Universal Robots URScript: A_penguin.script

def draw_penguin():
  # --- Robot Setup (ADJUST THESE VALUES) ---
  # Base position for the drawing (e.g., center of the A4 paper in robot's reach)
  base_p = p[0.4, -0.2, 0.2, 2.22, -2.22, 0]

  # Set the TCP for your marker tip. E.g., p[0, 0, 0.15, 0, 0, 0] for a 15cm offset
  # set_tcp(p[0, 0, 0.15, 0, 0, 0])

  # Movement parameters
  vel = 0.075
  accel = 0.1

  # Z heights for drawing (on paper) and moving (lifted)
  z_draw = base_p[2] - 0.005 # Adjust this based on paper height
  z_move = base_p[2] + 0.020 # 2cm lift

  # --- Drawing Logic ---
  textmsg("Starting the drawing process")
\n  # --- Path 1 ---\n  movel(pose(base_p[0] + 0.16907999999999998, base_p[1] + 0.024779999999999986, z_move, base_p[3], base_p[4], base_p[5]), a=accel, v=vel)\n  movel(pose(base_p[0] + 0.16907999999999998, base_p[1] + 0.024779999999999986, z_draw, base_p[3], base_p[4], base_p[5]), a=accel, v=vel)\n  movel(pose(base_p[0] + 0.1716, base_p[1] + 0.024779999999999986, z_draw, base_p[3], base_p[4], base_p[5]), a=accel, v=vel)\n  movel(pose(base_p[0] + 0.1716, base_p[1] + 0.024779999999999986, z_move, base_p[3], base_p[4], base_p[5]), a=accel, v=vel)\n\n  # --- Path 2 ---\n  movel(pose(base_p[0] + 0.18419999999999997, base_p[1] + 0.025619999999999987, z_move, base_p[3], base_p[4], base_p[5]), a=accel, v=vel)\n  movel(pose(base_p[0] + 0.18419999999999997, base_p[1] + 0.025619999999999987, z_draw, base_p[3], base_p[4], base_p[5]), a=accel, v=vel)\n  movel(pose(base_p[0] + 0.18336000000000002, base_p[1] + 0.024779999999999986, z_draw, base_p[3], base_p[4], base_p[5]), a=accel, v=vel)\n  movel(pose(base_p[0] + 0.18084, base_p[1] + 0.024779999999999986, z_draw, base_p[3], base_p[4], base_p[5]), a=accel, v=vel)\n  movel(pose(base_p[0] + 0.18419999999999997, base_p[1] + 0.024779999999999986, z_draw, base_p[3], base_p[4], base_p[5]), a=accel, v=vel)\n  movel(pose(base_p[0] + 0.18419999999999997, base_p[1] + 0.024779999999999986, z_move, base_p[3], base_p[4], base_p[5]), a=accel, v=vel)\n\n  # --- Path 3 ---\n  movel(pose(base_p[0] + 0.11279999999999998, base_p[1] + 0.025619999999999987, z_move, base_p[3], base_p[4], base_p[5]), a=accel, v=vel)\n  movel(pose(base_p[0] + 0.11279999999999998, base_p[1] + 0.025619999999999987, z_draw, base_p[3], base_p[4], base_p[5]), a=accel, v=vel)\n  movel(pose(base_p[0] + 0.11279999999999998, base_p[1] + 0.024779999999999986, z_draw, base_p[3], base_p[4], base_p[5]), a=accel, v=vel)\n  movel(pose(base_p[0] + 0.11363999999999999, base_p[1] + 0.023939999999999986, z_draw, base_p[3], base_p[4], base_p[5]), a=accel, v=vel)\n  movel(pose(base_p[0] + 0.11447999999999998, base_p[1] + 0.024779999999999986, z_draw, base_p[3], base_p[4], base_p[5]), a=accel, v=vel)\n  movel(pose(base_p[0] + 0.11616, base_p[1] + 0.024779999999999986, z_draw, base_p[3], base_p[4], base_p[5]), a=accel, v=vel)\n  movel(pose(base_p[0] + 0.11363999999999999, base_p[1] + 0.024779999999999986, z_draw, base_p[3], base_p[4], base_p[5]), a=accel, v=vel)\n  movel(pose(base_p[0] + 0.11363999999999999, base_p[1] + 0.024779999999999986, z_move, base_p[3], base_p[4], base_p[5]), a=accel, v=vel)\n\n  # --- Path 4 ---\n  movel(pose(base_p[0] + 0.16572, base_p[1] + 0.03401999999999999, z_move, base_p[3], base_p[4], base_p[5]), a=accel, v=vel)\n  movel(pose(base_p[0] + 0.16572, base_p[1] + 0.03401999999999999, z_draw, base_p[3], base_p[4], base_p[5]), a=accel, v=vel)\n  movel(pose(base_p[0] + 0.16656, base_p[1] + 0.033179999999999994, z_draw, base_p[3], base_p[4], base_p[5]), a=accel, v=vel)\n  movel(pose(base_p[0] + 0.17244, base_p[1] + 0.033179999999999994, z_draw, base_p[3], base_p[4], base_p[5]), a=accel, v=vel)\n  movel(pose(base_p[0] + 0.17244, base_p[1] + 0.03401999999999999, z_draw, base_p[3], base_p[4], base_p[5]), a=accel, v=vel)\n  movel(pose(base_p[0] + 0.1716, base_p[1] + 0.033179999999999994, z_draw, base_p[3], base_p[4], base_p[5]), a=accel, v=vel)\n  movel(pose(base_p[0] + 0.16739999999999997, base_p[1] + 0.033179999999999994, z_draw, base_p[3], base_p[4], base_p[5]), a=accel, v=vel)\n  movel(pose(base_p[0] + 0.16656, base_p[1] + 0.03401999999999999, z_draw, base_p[3], base_p[4], base_p[5]), a=accel, v=vel)\n  movel(pose(base_p[0] + 0.16824, base_p[1] + 0.03569999999999999, z_draw, base_p[3], base_p[4], base_p[5]), a=accel, v=vel)\n  movel(pose(base_p[0] + 0.16992000000000002, base_p[1] + 0.03569999999999999, z_draw, base_p[3], base_p[4], base_p[5]), a=accel, v=vel)\n  movel(pose(base_p[0] + 0.17076, base_p[1] + 0.03485999999999999, z_draw, base_p[3], base_p[4], base_p[5]), a=accel, v=vel)\n  movel(pose(base_p[0] + 0.1716, base_p[1] + 0.03569999999999999, z_draw, base_p[3], base_p[4], base_p[5]), a=accel, v=vel)\n  movel(pose(base_p[0] + 0.17412, base_p[1] + 0.03569999999999999, z_draw, base_p[3], base_p[4], base_p[5]), a=accel, v=vel)\n  movel(pose(base_p[0] + 0.16824, base_p[1] + 0.03569999999999999, z_draw, base_p[3], base_p[4], base_p[5]), a=accel, v=vel)\n  movel(pose(base_p[0] + 0.16739999999999997, base_p[1] + 0.03485999999999999, z_draw, base_p[3], base_p[4], base_p[5]), a=accel, v=vel)\n  movel(pose(base_p[0] + 0.16656, base_p[1] + 0.03485999999999999, z_draw, base_p[3], base_p[4], base_p[5]), a=accel, v=vel)\n  movel(pose(base_p[0] + 0.16656, base_p[1] + 0.03485999999999999, z_move, base_p[3], base_p[4], base_p[5]), a=accel, v=vel)\n\n  # --- Path 5 ---\n  movel(pose(base_p[0] + 0.12372, base_p[1] + 0.03653999999999999, z_move, base_p[3], base_p[4], base_p[5]), a=accel, v=vel)\n  movel(pose(base_p[0] + 0.12372, base_p[1] + 0.03653999999999999, z_draw, base_p[3], base_p[4], base_p[5]), a=accel, v=vel)\n  movel(pose(base_p[0] + 0.12455999999999999, base_p[1] + 0.03569999999999999, z_draw, base_p[3], base_p[4], base_p[5]), a=accel, v=vel)\n  movel(pose(base_p[0] + 0.12624, base_p[1] + 0.03569999999999999, z_draw, base_p[3], base_p[4], base_p[5]), a=accel, v=vel)\n  movel(pose(base_p[0] + 0.12708, base_p[1] + 0.03485999999999999, z_draw, base_p[3], base_p[4], base_p[5]), a=accel, v=vel)\n  movel(pose(base_p[0] + 0.1296, base_p[1] + 0.03485999999999999, z_draw, base_p[3], base_p[4], base_p[5]), a=accel, v=vel)\n  movel(pose(base_p[0] + 0.13127999999999998, base_p[1] + 0.033179999999999994, z_draw, base_p[3], base_p[4], base_p[5]), a=accel, v=vel)\n  movel(pose(base_p[0] + 0.13044, base_p[1] + 0.03233999999999999, z_draw, base_p[3], base_p[4], base_p[5]), a=accel, v=vel)\n  movel(pose(base_p[0] + 0.12791999999999998, base_p[1] + 0.03233999999999999, z_draw, base_p[3], base_p[4], base_p[5]), a=accel, v=vel)\n  movel(pose(base_p[0] + 0.12708, base_p[1] + 0.033179999999999994, z_draw, base_p[3], base_p[4], base_p[5]), a=accel, v=vel)\n  movel(pose(base_p[0] + 0.12624, base_p[1] + 0.03233999999999999, z_draw, base_p[3], base_p[4], base_p[5]), a=accel, v=vel)\n  movel(pose(base_p[0] + 0.12539999999999998, base_p[1] + 0.033179999999999994, z_draw, base_p[3], base_p[4], base_p[5]), a=accel, v=vel)\n  movel(pose(base_p[0] + 0.12455999999999999, base_p[1] + 0.033179999999999994, z_draw, base_p[3], base_p[4], base_p[5]), a=accel, v=vel)\n  movel(pose(base_p[0] + 0.12539999999999998, base_p[1] + 0.033179999999999994, z_draw, base_p[3], base_p[4], base_p[5]), a=accel, v=vel)\n  movel(pose(base_p[0] + 0.12624, base_p[1] + 0.03233999999999999, z_draw, base_p[3], base_p[4], base_p[5]), a=accel, v=vel)\n  movel(pose(base_p[0] + 0.12708, base_p[1] + 0.033179999999999994, z_draw, base_p[3], base_p[4], base_p[5]), a=accel, v=vel)\n  movel(pose(base_p[0] + 0.12791999999999998, base_p[1] + 0.03233999999999999, z_draw, base_p[3], base_p[4], base_p[5]), a=accel, v=vel)\n  movel(pose(base_p[0] + 0.13127999999999998, base_p[1] + 0.03233999999999999, z_draw, base_p[3], base_p[4], base_p[5]), a=accel, v=vel)\n  movel(pose(base_p[0] + 0.13127999999999998, base_p[1] + 0.03401999999999999, z_draw, base_p[3], base_p[4], base_p[5]), a=accel, v=vel)\n  movel(pose(base_p[0] + 0.13044, base_p[1] + 0.03401999999999999, z_draw, base_p[3], base_p[4], base_p[5]), a=accel, v=vel)\n  movel(pose(base_p[0] + 0.1296, base_p[1] + 0.03485999999999999, z_draw, base_p[3], base_p[4], base_p[5]), a=accel, v=vel)\n  movel(pose(base_p[0] + 0.12708, base_p[1] + 0.03485999999999999, z_draw, base_p[3], base_p[4], base_p[5]), a=accel, v=vel)\n  movel(pose(base_p[0] + 0.12624, base_p[1] + 0.03569999999999999, z_draw, base_p[3], base_p[4], base_p[5]), a=accel, v=vel)\n  movel(pose(base_p[0] + 0.12539999999999998, base_p[1] + 0.03569999999999999, z_draw, base_p[3], base_p[4], base_p[5]), a=accel, v=vel)\n  movel(pose(base_p[0] + 0.12455999999999999, base_p[1] + 0.03653999999999999, z_draw, base_p[3], base_p[4], base_p[5]), a=accel, v=vel)\n  movel(pose(base_p[0] + 0.12455999999999999, base_p[1] + 0.03653999999999999, z_move, base_p[3], base_p[4], base_p[5]), a=accel, v=vel)\n\n  # --- Path 6 ---\n  movel(pose(base_p[0] + 0.13883999999999996, base_p[1] + 0.040739999999999985, z_move, base_p[3], base_p[4], base_p[5]), a=accel, v=vel)\n  movel(pose(base_p[0] + 0.13883999999999996, base_p[1] + 0.040739999999999985, z_draw, base_p[3], base_p[4], base_p[5]), a=accel, v=vel)\n  movel(pose(base_p[0] + 0.13968, base_p[1] + 0.03989999999999999, z_draw, base_p[3], base_p[4], base_p[5]), a=accel, v=vel)\n  movel(pose(base_p[0] + 0.13968, base_p[1] + 0.03905999999999999, z_draw, base_p[3], base_p[4], base_p[5]), a=accel, v=vel)\n  movel(pose(base_p[0] + 0.14051999999999998, base_p[1] + 0.03905999999999999, z_draw, base_p[3], base_p[4], base_p[5]), a=accel, v=vel)\n  movel(pose(base_p[0] + 0.14136, base_p[1] + 0.03821999999999998, z_draw, base_p[3], base_p[4], base_p[5]), a=accel, v=vel)\n  movel(pose(base_p[0] + 0.14304, base_p[1] + 0.03821999999999998, z_draw, base_p[3], base_p[4], base_p[5]), a=accel, v=vel)\n  movel(pose(base_p[0] + 0.14388, base_p[1] + 0.03737999999999999, z_draw, base_p[3], base_p[4], base_p[5]), a=accel, v=vel)\n  movel(pose(base_p[0] + 0.14472, base_p[1] + 0.03737999999999999, z_draw, base_p[3], base_p[4], base_p[5]), a=accel, v=vel)\n  movel(pose(base_p[0] + 0.14556, base_p[1] + 0.03653999999999999, z_draw, base_p[3], base_p[4], base_p[5]), a=accel, v=vel)\n  movel(pose(base_p[0] + 0.14639999999999997, base_p[1] + 0.03737999999999999, z_draw, base_p[3], base_p[4], base_p[5]), a=accel, v=vel)\n  movel(pose(base_p[0] + 0.14724, base_p[1] + 0.03737999999999999, z_draw, base_p[3], base_p[4], base_p[5]), a=accel, v=vel)\n  movel(pose(base_p[0] + 0.14808, base_p[1] + 0.03653999999999999, z_draw, base_p[3], base_p[4], base_p[5]), a=accel, v=vel)\n  movel(pose(base_p[0] + 0.14976, base_p[1] + 0.03653999999999999, z_draw, base_p[3], base_p[4], base_p[5]), a=accel, v=vel)\n  movel(pose(base_p[0] + 0.15059999999999998, base_p[1] + 0.03737999999999999, z_draw, base_p[3], base_p[4], base_p[5]), a=accel, v=vel)\n  movel(pose(base_p[0] + 0.15228, base_p[1] + 0.03737999999999999, z_draw, base_p[3], base_p[4], base_p[5]), a=accel, v=vel)\n  movel(pose(base_p[0] + 0.15312, base_p[1] + 0.03821999999999998, z_draw, base_p[3], base_p[4], base_p[5]), a=accel, v=vel)\n  movel(pose(base_p[0] + 0.15395999999999999, base_p[1] + 0.03821999999999998, z_draw, base_p[3], base_p[4], base_p[5]), a=accel, v=vel)\n  movel(pose(base_p[0] + 0.15480000000000002, base_p[1] + 0.03905999999999999, z_draw, base_p[3], base_p[4], base_p[5]), a=accel, v=vel)\n  movel(pose(base_p[0] + 0.15563999999999997, base_p[1] + 0.03905999999999999, z_draw, base_p[3], base_p[4], base_p[5]), a=accel, v=vel)\n  movel(pose(base_p[0] + 0.15647999999999998, base_p[1] + 0.03989999999999999, z_draw, base_p[3], base_p[4], base_p[5]), a=accel, v=vel)\n  movel(pose(base_p[0] + 0.15563999999999997, base_p[1] + 0.03989999999999999, z_draw, base_p[3], base_p[4], base_p[5]), a=accel, v=vel)\n  movel(pose(base_p[0] + 0.15480000000000002, base_p[1] + 0.03905999999999999, z_draw, base_p[3], base_p[4], base_p[5]), a=accel, v=vel)\n  movel(pose(base_p[0] + 0.15395999999999999, base_p[1] + 0.03905999999999999, z_draw, base_p[3], base_p[4], base_p[5]), a=accel, v=vel)\n  movel(pose(base_p[0] + 0.15228, base_p[1] + 0.03737999999999999, z_draw, base_p[3], base_p[4], base_p[5]), a=accel, v=vel)\n  movel(pose(base_p[0] + 0.15059999999999998, base_p[1] + 0.03737999999999999, z_draw, base_p[3], base_p[4], base_p[5]), a=accel, v=vel)\n  movel(pose(base_p[0] + 0.14976, base_p[1] + 0.03653999999999999, z_draw, base_p[3], base_p[4], base_p[5]), a=accel, v=vel)\n  movel(pose(base_p[0] + 0.14808, base_p[1] + 0.03653999999999999, z_draw, base_p[3], base_p[4], base_p[5]), a=accel, v=vel)\n  movel(pose(base_p[0] + 0.14724, base_p[1] + 0.03737999999999999, z_draw, base_p[3], base_p[4], base_p[5]), a=accel, v=vel)\n  movel(pose(base_p[0] + 0.14472, base_p[1] + 0.03737999999999999, z_draw, base_p[3], base_p[4], base_p[5]), a=accel, v=vel)\n  movel(pose(base_p[0] + 0.14388, base_p[1] + 0.03821999999999998, z_draw, base_p[3], base_p[4], base_p[5]), a=accel, v=vel)\n  movel(pose(base_p[0] + 0.14136, base_p[1] + 0.03821999999999998, z_draw, base_p[3], base_p[4], base_p[5]), a=accel, v=vel)\n  movel(pose(base_p[0] + 0.13968, base_p[1] + 0.03989999999999999, z_draw, base_p[3], base_p[4], base_p[5]), a=accel, v=vel)\n  movel(pose(base_p[0] + 0.13968, base_p[1] + 0.040739999999999985, z_draw, base_p[3], base_p[4], base_p[5]), a=accel, v=vel)\n  movel(pose(base_p[0] + 0.13968, base_p[1] + 0.040739999999999985, z_move, base_p[3], base_p[4], base_p[5]), a=accel, v=vel)\n\n  # --- Path 7 ---\n  movel(pose(base_p[0] + 0.09348, base_p[1] + 0.11045999999999999, z_move, base_p[3], base_p[4], base_p[5]), a=accel, v=vel)\n  movel(pose(base_p[0] + 0.09348, base_p[1] + 0.11045999999999999, z_draw, base_p[3], base_p[4], base_p[5]), a=accel, v=vel)\n  movel(pose(base_p[0] + 0.09011999999999999, base_p[1] + 0.10878, z_draw, base_p[3], base_p[4], base_p[5]), a=accel, v=vel)\n  movel(pose(base_p[0] + 0.08675999999999999, base_p[1] + 0.10542, z_draw, base_p[3], base_p[4], base_p[5]), a=accel, v=vel)\n  movel(pose(base_p[0] + 0.08591999999999998, base_p[1] + 0.10289999999999999, z_draw, base_p[3], base_p[4], base_p[5]), a=accel, v=vel)\n  movel(pose(base_p[0] + 0.07919999999999999, base_p[1] + 0.09617999999999999, z_draw, base_p[3], base_p[4], base_p[5]), a=accel, v=vel)\n  movel(pose(base_p[0] + 0.07835999999999999, base_p[1] + 0.09617999999999999, z_draw, base_p[3], base_p[4], base_p[5]), a=accel, v=vel)\n  movel(pose(base_p[0] + 0.07499999999999998, base_p[1] + 0.09029999999999999, z_draw, base_p[3], base_p[4], base_p[5]), a=accel, v=vel)\n  movel(pose(base_p[0] + 0.07247999999999999, base_p[1] + 0.08777999999999998, z_draw, base_p[3], base_p[4], base_p[5]), a=accel, v=vel)\n  movel(pose(base_p[0] + 0.06828, base_p[1] + 0.07937999999999999, z_draw, base_p[3], base_p[4], base_p[5]), a=accel, v=vel)\n  movel(pose(base_p[0] + 0.06828, base_p[1] + 0.07769999999999999, z_draw, base_p[3], base_p[4], base_p[5]), a=accel, v=vel)\n  movel(pose(base_p[0] + 0.07247999999999999, base_p[1] + 0.08694, z_draw, base_p[3], base_p[4], base_p[5]), a=accel, v=vel)\n  movel(pose(base_p[0] + 0.07499999999999998, base_p[1] + 0.08946, z_draw, base_p[3], base_p[4], base_p[5]), a=accel, v=vel)\n  movel(pose(base_p[0] + 0.07751999999999998, base_p[1] + 0.0945, z_draw, base_p[3], base_p[4], base_p[5]), a=accel, v=vel)\n  movel(pose(base_p[0] + 0.07919999999999999, base_p[1] + 0.09617999999999999, z_draw, base_p[3], base_p[4], base_p[5]), a=accel, v=vel)\n  movel(pose(base_p[0] + 0.08003999999999999, base_p[1] + 0.09617999999999999, z_draw, base_p[3], base_p[4], base_p[5]), a=accel, v=vel)\n  movel(pose(base_p[0] + 0.08591999999999998, base_p[1] + 0.10205999999999998, z_draw, base_p[3], base_p[4], base_p[5]), a=accel, v=vel)\n  movel(pose(base_p[0] + 0.08675999999999999, base_p[1] + 0.10457999999999999, z_draw, base_p[3], base_p[4], base_p[5]), a=accel, v=vel)\n  movel(pose(base_p[0] + 0.09263999999999999, base_p[1] + 0.11045999999999999, z_draw, base_p[3], base_p[4], base_p[5]), a=accel, v=vel)\n  movel(pose(base_p[0] + 0.09263999999999999, base_p[1] + 0.11045999999999999, z_move, base_p[3], base_p[4], base_p[5]), a=accel, v=vel)\n\n  # --- Path 8 ---\n  movel(pose(base_p[0] + 0.11279999999999998, base_p[1] + 0.1281, z_move, base_p[3], base_p[4], base_p[5]), a=accel, v=vel)\n  movel(pose(base_p[0] + 0.11279999999999998, base_p[1] + 0.1281, z_draw, base_p[3], base_p[4], base_p[5]), a=accel, v=vel)\n  movel(pose(base_p[0] + 0.11112, base_p[1] + 0.12642, z_draw, base_p[3], base_p[4], base_p[5]), a=accel, v=vel)\n  movel(pose(base_p[0] + 0.11028, base_p[1] + 0.12642, z_draw, base_p[3], base_p[4], base_p[5]), a=accel, v=vel)\n  movel(pose(base_p[0] + 0.10859999999999999, base_p[1] + 0.12473999999999999, z_draw, base_p[3], base_p[4], base_p[5]), a=accel, v=vel)\n  movel(pose(base_p[0] + 0.10859999999999999, base_p[1] + 0.1239, z_draw, base_p[3], base_p[4], base_p[5]), a=accel, v=vel)\n  movel(pose(base_p[0] + 0.11112, base_p[1] + 0.12642, z_draw, base_p[3], base_p[4], base_p[5]), a=accel, v=vel)\n  movel(pose(base_p[0] + 0.11195999999999999, base_p[1] + 0.12642, z_draw, base_p[3], base_p[4], base_p[5]), a=accel, v=vel)\n  movel(pose(base_p[0] + 0.11279999999999998, base_p[1] + 0.12725999999999998, z_draw, base_p[3], base_p[4], base_p[5]), a=accel, v=vel)\n  movel(pose(base_p[0] + 0.11279999999999998, base_p[1] + 0.12725999999999998, z_move, base_p[3], base_p[4], base_p[5]), a=accel, v=vel)\n\n  # --- Path 9 ---\n  movel(pose(base_p[0] + 0.12119999999999999, base_p[1] + 0.13062, z_move, base_p[3], base_p[4], base_p[5]), a=accel, v=vel)\n  movel(pose(base_p[0] + 0.12119999999999999, base_p[1] + 0.13062, z_draw, base_p[3], base_p[4], base_p[5]), a=accel, v=vel)\n  movel(pose(base_p[0] + 0.12119999999999999, base_p[1] + 0.12725999999999998, z_draw, base_p[3], base_p[4], base_p[5]), a=accel, v=vel)\n  movel(pose(base_p[0] + 0.12204, base_p[1] + 0.12642, z_draw, base_p[3], base_p[4], base_p[5]), a=accel, v=vel)\n  movel(pose(base_p[0] + 0.12119999999999999, base_p[1] + 0.12558, z_draw, base_p[3], base_p[4], base_p[5]), a=accel, v=vel)\n  movel(pose(base_p[0] + 0.12119999999999999, base_p[1] + 0.12138, z_draw, base_p[3], base_p[4], base_p[5]), a=accel, v=vel)\n  movel(pose(base_p[0] + 0.12035999999999998, base_p[1] + 0.12054, z_draw, base_p[3], base_p[4], base_p[5]), a=accel, v=vel)\n  movel(pose(base_p[0] + 0.12035999999999998, base_p[1] + 0.11717999999999999, z_draw, base_p[3], base_p[4], base_p[5]), a=accel, v=vel)\n  movel(pose(base_p[0] + 0.11868, base_p[1] + 0.1155, z_draw, base_p[3], base_p[4], base_p[5]), a=accel, v=vel)\n  movel(pose(base_p[0] + 0.11868, base_p[1] + 0.11466, z_draw, base_p[3], base_p[4], base_p[5]), a=accel, v=vel)\n  movel(pose(base_p[0] + 0.11952, base_p[1] + 0.1155, z_draw, base_p[3], base_p[4], base_p[5]), a=accel, v=vel)\n  movel(pose(base_p[0] + 0.11952, base_p[1] + 0.11633999999999999, z_draw, base_p[3], base_p[4], base_p[5]), a=accel, v=vel)\n  movel(pose(base_p[0] + 0.12035999999999998, base_p[1] + 0.11717999999999999, z_draw, base_p[3], base_p[4], base_p[5]), a=accel, v=vel)\n  movel(pose(base_p[0] + 0.12035999999999998, base_p[1] + 0.12054, z_draw, base_p[3], base_p[4], base_p[5]), a=accel, v=vel)\n  movel(pose(base_p[0] + 0.12119999999999999, base_p[1] + 0.12138, z_draw, base_p[3], base_p[4], base_p[5]), a=accel, v=vel)\n  movel(pose(base_p[0] + 0.12119999999999999, base_p[1] + 0.12558, z_draw, base_p[3], base_p[4], base_p[5]), a=accel, v=vel)\n  movel(pose(base_p[0] + 0.12204, base_p[1] + 0.12642, z_draw, base_p[3], base_p[4], base_p[5]), a=accel, v=vel)\n  movel(pose(base_p[0] + 0.12119999999999999, base_p[1] + 0.12725999999999998, z_draw, base_p[3], base_p[4], base_p[5]), a=accel, v=vel)\n  movel(pose(base_p[0] + 0.12119999999999999, base_p[1] + 0.12725999999999998, z_move, base_p[3], base_p[4], base_p[5]), a=accel, v=vel)\n\n  # --- Path 10 ---\n  movel(pose(base_p[0] + 0.1338, base_p[1] + 0.15077999999999997, z_move, base_p[3], base_p[4], base_p[5]), a=accel, v=vel)\n  movel(pose(base_p[0] + 0.1338, base_p[1] + 0.15077999999999997, z_draw, base_p[3], base_p[4], base_p[5]), a=accel, v=vel)\n  movel(pose(base_p[0] + 0.13463999999999998, base_p[1] + 0.14826, z_draw, base_p[3], base_p[4], base_p[5]), a=accel, v=vel)\n  movel(pose(base_p[0] + 0.138, base_p[1] + 0.14658, z_draw, base_p[3], base_p[4], base_p[5]), a=accel, v=vel)\n  movel(pose(base_p[0] + 0.14639999999999997, base_p[1] + 0.14574, z_draw, base_p[3], base_p[4], base_p[5]), a=accel, v=vel)\n  movel(pose(base_p[0] + 0.14724, base_p[1] + 0.14489999999999997, z_draw, base_p[3], base_p[4], base_p[5]), a=accel, v=vel)\n  movel(pose(base_p[0] + 0.15480000000000002, base_p[1] + 0.14574, z_draw, base_p[3], base_p[4], base_p[5]), a=accel, v=vel)\n  movel(pose(base_p[0] + 0.16236, base_p[1] + 0.14826, z_draw, base_p[3], base_p[4], base_p[5]), a=accel, v=vel)\n  movel(pose(base_p[0] + 0.15983999999999998, base_p[1] + 0.14826, z_draw, base_p[3], base_p[4], base_p[5]), a=accel, v=vel)\n  movel(pose(base_p[0] + 0.15480000000000002, base_p[1] + 0.14574, z_draw, base_p[3], base_p[4], base_p[5]), a=accel, v=vel)\n  movel(pose(base_p[0] + 0.14724, base_p[1] + 0.14489999999999997, z_draw, base_p[3], base_p[4], base_p[5]), a=accel, v=vel)\n  movel(pose(base_p[0] + 0.13632, base_p[1] + 0.14742000000000002, z_draw, base_p[3], base_p[4], base_p[5]), a=accel, v=vel)\n  movel(pose(base_p[0] + 0.1338, base_p[1] + 0.14994, z_draw, base_p[3], base_p[4], base_p[5]), a=accel, v=vel)\n  movel(pose(base_p[0] + 0.13463999999999998, base_p[1] + 0.15077999999999997, z_draw, base_p[3], base_p[4], base_p[5]), a=accel, v=vel)\n  movel(pose(base_p[0] + 0.14388, base_p[1] + 0.14742000000000002, z_draw, base_p[3], base_p[4], base_p[5]), a=accel, v=vel)\n  movel(pose(base_p[0] + 0.15228, base_p[1] + 0.14742000000000002, z_draw, base_p[3], base_p[4], base_p[5]), a=accel, v=vel)\n  movel(pose(base_p[0] + 0.159, base_p[1] + 0.14994, z_draw, base_p[3], base_p[4], base_p[5]), a=accel, v=vel)\n  movel(pose(base_p[0] + 0.16236, base_p[1] + 0.14994, z_draw, base_p[3], base_p[4], base_p[5]), a=accel, v=vel)\n  movel(pose(base_p[0] + 0.159, base_p[1] + 0.14994, z_draw, base_p[3], base_p[4], base_p[5]), a=accel, v=vel)\n  movel(pose(base_p[0] + 0.15228, base_p[1] + 0.14742000000000002, z_draw, base_p[3], base_p[4], base_p[5]), a=accel, v=vel)\n  movel(pose(base_p[0] + 0.14388, base_p[1] + 0.14742000000000002, z_draw, base_p[3], base_p[4], base_p[5]), a=accel, v=vel)\n  movel(pose(base_p[0] + 0.138, base_p[1] + 0.1491, z_draw, base_p[3], base_p[4], base_p[5]), a=accel, v=vel)\n  movel(pose(base_p[0] + 0.13632, base_p[1] + 0.15077999999999997, z_draw, base_p[3], base_p[4], base_p[5]), a=accel, v=vel)\n  movel(pose(base_p[0] + 0.13632, base_p[1] + 0.15077999999999997, z_move, base_p[3], base_p[4], base_p[5]), a=accel, v=vel)\n\n  # --- Path 11 ---\n  movel(pose(base_p[0] + 0.13883999999999996, base_p[1] + 0.16506, z_move, base_p[3], base_p[4], base_p[5]), a=accel, v=vel)\n  movel(pose(base_p[0] + 0.13883999999999996, base_p[1] + 0.16506, z_draw, base_p[3], base_p[4], base_p[5]), a=accel, v=vel)\n  movel(pose(base_p[0] + 0.13968, base_p[1] + 0.16589999999999996, z_draw, base_p[3], base_p[4], base_p[5]), a=accel, v=vel)\n  movel(pose(base_p[0] + 0.14051999999999998, base_p[1] + 0.16506, z_draw, base_p[3], base_p[4], base_p[5]), a=accel, v=vel)\n  movel(pose(base_p[0] + 0.13968, base_p[1] + 0.16422000000000003, z_draw, base_p[3], base_p[4], base_p[5]), a=accel, v=vel)\n  movel(pose(base_p[0] + 0.13968, base_p[1] + 0.16422000000000003, z_move, base_p[3], base_p[4], base_p[5]), a=accel, v=vel)\n\n  # --- Path 12 ---\n  movel(pose(base_p[0] + 0.14808, base_p[1] + 0.16926, z_move, base_p[3], base_p[4], base_p[5]), a=accel, v=vel)\n  movel(pose(base_p[0] + 0.14808, base_p[1] + 0.16926, z_draw, base_p[3], base_p[4], base_p[5]), a=accel, v=vel)\n  movel(pose(base_p[0] + 0.14892000000000002, base_p[1] + 0.16926, z_draw, base_p[3], base_p[4], base_p[5]), a=accel, v=vel)\n  movel(pose(base_p[0] + 0.15312, base_p[1] + 0.16506, z_draw, base_p[3], base_p[4], base_p[5]), a=accel, v=vel)\n  movel(pose(base_p[0] + 0.14976, base_p[1] + 0.16169999999999998, z_draw, base_p[3], base_p[4], base_p[5]), a=accel, v=vel)\n  movel(pose(base_p[0] + 0.14808, base_p[1] + 0.16169999999999998, z_draw, base_p[3], base_p[4], base_p[5]), a=accel, v=vel)\n  movel(pose(base_p[0] + 0.14724, base_p[1] + 0.16254000000000002, z_draw, base_p[3], base_p[4], base_p[5]), a=accel, v=vel)\n  movel(pose(base_p[0] + 0.14639999999999997, base_p[1] + 0.16254000000000002, z_draw, base_p[3], base_p[4], base_p[5]), a=accel, v=vel)\n  movel(pose(base_p[0] + 0.14556, base_p[1] + 0.16338, z_draw, base_p[3], base_p[4], base_p[5]), a=accel, v=vel)\n  movel(pose(base_p[0] + 0.14556, base_p[1] + 0.16422000000000003, z_draw, base_p[3], base_p[4], base_p[5]), a=accel, v=vel)\n  movel(pose(base_p[0] + 0.14472, base_p[1] + 0.16506, z_draw, base_p[3], base_p[4], base_p[5]), a=accel, v=vel)\n  movel(pose(base_p[0] + 0.14556, base_p[1] + 0.16589999999999996, z_draw, base_p[3], base_p[4], base_p[5]), a=accel, v=vel)\n  movel(pose(base_p[0] + 0.14556, base_p[1] + 0.16674, z_draw, base_p[3], base_p[4], base_p[5]), a=accel, v=vel)\n  movel(pose(base_p[0] + 0.14556, base_p[1] + 0.16674, z_move, base_p[3], base_p[4], base_p[5]), a=accel, v=vel)\n\n  # --- Path 13 ---\n  movel(pose(base_p[0] + 0.14724, base_p[1] + 0.16926, z_move, base_p[3], base_p[4], base_p[5]), a=accel, v=vel)\n  movel(pose(base_p[0] + 0.14724, base_p[1] + 0.16926, z_draw, base_p[3], base_p[4], base_p[5]), a=accel, v=vel)\n  movel(pose(base_p[0] + 0.14556, base_p[1] + 0.16757999999999998, z_draw, base_p[3], base_p[4], base_p[5]), a=accel, v=vel)\n  movel(pose(base_p[0] + 0.14556, base_p[1] + 0.16674, z_draw, base_p[3], base_p[4], base_p[5]), a=accel, v=vel)\n  movel(pose(base_p[0] + 0.14472, base_p[1] + 0.16589999999999996, z_draw, base_p[3], base_p[4], base_p[5]), a=accel, v=vel)\n  movel(pose(base_p[0] + 0.14472, base_p[1] + 0.16422000000000003, z_draw, base_p[3], base_p[4], base_p[5]), a=accel, v=vel)\n  movel(pose(base_p[0] + 0.14556, base_p[1] + 0.16338, z_draw, base_p[3], base_p[4], base_p[5]), a=accel, v=vel)\n  movel(pose(base_p[0] + 0.14556, base_p[1] + 0.16254000000000002, z_draw, base_p[3], base_p[4], base_p[5]), a=accel, v=vel)\n  movel(pose(base_p[0] + 0.14639999999999997, base_p[1] + 0.16254000000000002, z_draw, base_p[3], base_p[4], base_p[5]), a=accel, v=vel)\n  movel(pose(base_p[0] + 0.14724, base_p[1] + 0.16169999999999998, z_draw, base_p[3], base_p[4], base_p[5]), a=accel, v=vel)\n  movel(pose(base_p[0] + 0.15059999999999998, base_p[1] + 0.16169999999999998, z_draw, base_p[3], base_p[4], base_p[5]), a=accel, v=vel)\n  movel(pose(base_p[0] + 0.15144, base_p[1] + 0.16254000000000002, z_draw, base_p[3], base_p[4], base_p[5]), a=accel, v=vel)\n  movel(pose(base_p[0] + 0.15144, base_p[1] + 0.16338, z_draw, base_p[3], base_p[4], base_p[5]), a=accel, v=vel)\n  movel(pose(base_p[0] + 0.15312, base_p[1] + 0.16506, z_draw, base_p[3], base_p[4], base_p[5]), a=accel, v=vel)\n  movel(pose(base_p[0] + 0.15395999999999999, base_p[1] + 0.16506, z_draw, base_p[3], base_p[4], base_p[5]), a=accel, v=vel)\n  movel(pose(base_p[0] + 0.14976, base_p[1] + 0.16926, z_draw, base_p[3], base_p[4], base_p[5]), a=accel, v=vel)\n  movel(pose(base_p[0] + 0.14976, base_p[1] + 0.16926, z_move, base_p[3], base_p[4], base_p[5]), a=accel, v=vel)\n\n  # --- Path 14 ---\n  movel(pose(base_p[0] + 0.16236, base_p[1] + 0.17178000000000002, z_move, base_p[3], base_p[4], base_p[5]), a=accel, v=vel)\n  movel(pose(base_p[0] + 0.16236, base_p[1] + 0.17178000000000002, z_draw, base_p[3], base_p[4], base_p[5]), a=accel, v=vel)\n  movel(pose(base_p[0] + 0.16404, base_p[1] + 0.17010000000000003, z_draw, base_p[3], base_p[4], base_p[5]), a=accel, v=vel)\n  movel(pose(base_p[0] + 0.16404, base_p[1] + 0.16842000000000001, z_draw, base_p[3], base_p[4], base_p[5]), a=accel, v=vel)\n  movel(pose(base_p[0] + 0.16236, base_p[1] + 0.16674, z_draw, base_p[3], base_p[4], base_p[5]), a=accel, v=vel)\n  movel(pose(base_p[0] + 0.16151999999999997, base_p[1] + 0.16674, z_draw, base_p[3], base_p[4], base_p[5]), a=accel, v=vel)\n  movel(pose(base_p[0] + 0.16068000000000002, base_p[1] + 0.16757999999999998, z_draw, base_p[3], base_p[4], base_p[5]), a=accel, v=vel)\n  movel(pose(base_p[0] + 0.16068000000000002, base_p[1] + 0.16926, z_draw, base_p[3], base_p[4], base_p[5]), a=accel, v=vel)\n  movel(pose(base_p[0] + 0.16151999999999997, base_p[1] + 0.17010000000000003, z_draw, base_p[3], base_p[4], base_p[5]), a=accel, v=vel)\n  movel(pose(base_p[0] + 0.16151999999999997, base_p[1] + 0.17094, z_draw, base_p[3], base_p[4], base_p[5]), a=accel, v=vel)\n  movel(pose(base_p[0] + 0.16151999999999997, base_p[1] + 0.17094, z_move, base_p[3], base_p[4], base_p[5]), a=accel, v=vel)\n\n  # --- Path 15 ---\n  movel(pose(base_p[0] + 0.13463999999999998, base_p[1] + 0.17178000000000002, z_move, base_p[3], base_p[4], base_p[5]), a=accel, v=vel)\n  movel(pose(base_p[0] + 0.13463999999999998, base_p[1] + 0.17178000000000002, z_draw, base_p[3], base_p[4], base_p[5]), a=accel, v=vel)\n  movel(pose(base_p[0] + 0.13632, base_p[1] + 0.17010000000000003, z_draw, base_p[3], base_p[4], base_p[5]), a=accel, v=vel)\n  movel(pose(base_p[0] + 0.13632, base_p[1] + 0.16926, z_draw, base_p[3], base_p[4], base_p[5]), a=accel, v=vel)\n  movel(pose(base_p[0] + 0.13716, base_p[1] + 0.16842000000000001, z_draw, base_p[3], base_p[4], base_p[5]), a=accel, v=vel)\n  movel(pose(base_p[0] + 0.13548, base_p[1] + 0.16674, z_draw, base_p[3], base_p[4], base_p[5]), a=accel, v=vel)\n  movel(pose(base_p[0] + 0.13463999999999998, base_p[1] + 0.16674, z_draw, base_p[3], base_p[4], base_p[5]), a=accel, v=vel)\n  movel(pose(base_p[0] + 0.13295999999999997, base_p[1] + 0.16842000000000001, z_draw, base_p[3], base_p[4], base_p[5]), a=accel, v=vel)\n  movel(pose(base_p[0] + 0.13295999999999997, base_p[1] + 0.17010000000000003, z_draw, base_p[3], base_p[4], base_p[5]), a=accel, v=vel)\n  movel(pose(base_p[0] + 0.13295999999999997, base_p[1] + 0.17010000000000003, z_move, base_p[3], base_p[4], base_p[5]), a=accel, v=vel)\n\n  # --- Path 16 ---\n  movel(pose(base_p[0] + 0.16151999999999997, base_p[1] + 0.17178000000000002, z_move, base_p[3], base_p[4], base_p[5]), a=accel, v=vel)\n  movel(pose(base_p[0] + 0.16151999999999997, base_p[1] + 0.17178000000000002, z_draw, base_p[3], base_p[4], base_p[5]), a=accel, v=vel)\n  movel(pose(base_p[0] + 0.16151999999999997, base_p[1] + 0.17094, z_draw, base_p[3], base_p[4], base_p[5]), a=accel, v=vel)\n  movel(pose(base_p[0] + 0.16068000000000002, base_p[1] + 0.17010000000000003, z_draw, base_p[3], base_p[4], base_p[5]), a=accel, v=vel)\n  movel(pose(base_p[0] + 0.16068000000000002, base_p[1] + 0.16674, z_draw, base_p[3], base_p[4], base_p[5]), a=accel, v=vel)\n  movel(pose(base_p[0] + 0.16319999999999998, base_p[1] + 0.16674, z_draw, base_p[3], base_p[4], base_p[5]), a=accel, v=vel)\n  movel(pose(base_p[0] + 0.16404, base_p[1] + 0.16757999999999998, z_draw, base_p[3], base_p[4], base_p[5]), a=accel, v=vel)\n  movel(pose(base_p[0] + 0.16404, base_p[1] + 0.17094, z_draw, base_p[3], base_p[4], base_p[5]), a=accel, v=vel)\n  movel(pose(base_p[0] + 0.16319999999999998, base_p[1] + 0.17178000000000002, z_draw, base_p[3], base_p[4], base_p[5]), a=accel, v=vel)\n  movel(pose(base_p[0] + 0.16319999999999998, base_p[1] + 0.17178000000000002, z_move, base_p[3], base_p[4], base_p[5]), a=accel, v=vel)\n\n  # --- Path 17 ---\n  movel(pose(base_p[0] + 0.1338, base_p[1] + 0.17178000000000002, z_move, base_p[3], base_p[4], base_p[5]), a=accel, v=vel)\n  movel(pose(base_p[0] + 0.1338, base_p[1] + 0.17178000000000002, z_draw, base_p[3], base_p[4], base_p[5]), a=accel, v=vel)\n  movel(pose(base_p[0] + 0.13295999999999997, base_p[1] + 0.17094, z_draw, base_p[3], base_p[4], base_p[5]), a=accel, v=vel)\n  movel(pose(base_p[0] + 0.13295999999999997, base_p[1] + 0.16757999999999998, z_draw, base_p[3], base_p[4], base_p[5]), a=accel, v=vel)\n  movel(pose(base_p[0] + 0.1338, base_p[1] + 0.16674, z_draw, base_p[3], base_p[4], base_p[5]), a=accel, v=vel)\n  movel(pose(base_p[0] + 0.13632, base_p[1] + 0.16674, z_draw, base_p[3], base_p[4], base_p[5]), a=accel, v=vel)\n  movel(pose(base_p[0] + 0.13632, base_p[1] + 0.16757999999999998, z_draw, base_p[3], base_p[4], base_p[5]), a=accel, v=vel)\n  movel(pose(base_p[0] + 0.13716, base_p[1] + 0.16842000000000001, z_draw, base_p[3], base_p[4], base_p[5]), a=accel, v=vel)\n  movel(pose(base_p[0] + 0.13632, base_p[1] + 0.16926, z_draw, base_p[3], base_p[4], base_p[5]), a=accel, v=vel)\n  movel(pose(base_p[0] + 0.13632, base_p[1] + 0.17094, z_draw, base_p[3], base_p[4], base_p[5]), a=accel, v=vel)\n  movel(pose(base_p[0] + 0.13548, base_p[1] + 0.17094, z_draw, base_p[3], base_p[4], base_p[5]), a=accel, v=vel)\n  movel(pose(base_p[0] + 0.13463999999999998, base_p[1] + 0.17178000000000002, z_draw, base_p[3], base_p[4], base_p[5]), a=accel, v=vel)\n  movel(pose(base_p[0] + 0.13463999999999998, base_p[1] + 0.17178000000000002, z_move, base_p[3], base_p[4], base_p[5]), a=accel, v=vel)\n\n  # --- Path 18 ---\n  movel(pose(base_p[0] + 0.16068000000000002, base_p[1] + 0.17598000000000003, z_move, base_p[3], base_p[4], base_p[5]), a=accel, v=vel)\n  movel(pose(base_p[0] + 0.16068000000000002, base_p[1] + 0.17598000000000003, z_draw, base_p[3], base_p[4], base_p[5]), a=accel, v=vel)\n  movel(pose(base_p[0] + 0.15732, base_p[1] + 0.16589999999999996, z_draw, base_p[3], base_p[4], base_p[5]), a=accel, v=vel)\n  movel(pose(base_p[0] + 0.16151999999999997, base_p[1] + 0.17598000000000003, z_draw, base_p[3], base_p[4], base_p[5]), a=accel, v=vel)\n  movel(pose(base_p[0] + 0.16824, base_p[1] + 0.17010000000000003, z_draw, base_p[3], base_p[4], base_p[5]), a=accel, v=vel)\n  movel(pose(base_p[0] + 0.16992000000000002, base_p[1] + 0.16254000000000002, z_draw, base_p[3], base_p[4], base_p[5]), a=accel, v=vel)\n  movel(pose(base_p[0] + 0.16656, base_p[1] + 0.15245999999999998, z_draw, base_p[3], base_p[4], base_p[5]), a=accel, v=vel)\n  movel(pose(base_p[0] + 0.1716, base_p[1] + 0.14826, z_draw, base_p[3], base_p[4], base_p[5]), a=accel, v=vel)\n  movel(pose(base_p[0] + 0.18252, base_p[1] + 0.12558, z_draw, base_p[3], base_p[4], base_p[5]), a=accel, v=vel)\n  movel(pose(base_p[0] + 0.19007999999999997, base_p[1] + 0.08106, z_draw, base_p[3], base_p[4], base_p[5]), a=accel, v=vel)\n  movel(pose(base_p[0] + 0.18756, base_p[1] + 0.05165999999999999, z_draw, base_p[3], base_p[4], base_p[5]), a=accel, v=vel)\n  movel(pose(base_p[0] + 0.18168, base_p[1] + 0.041579999999999985, z_draw, base_p[3], base_p[4], base_p[5]), a=accel, v=vel)\n  movel(pose(base_p[0] + 0.17832, base_p[1] + 0.041579999999999985, z_draw, base_p[3], base_p[4], base_p[5]), a=accel, v=vel)\n  movel(pose(base_p[0] + 0.17412, base_p[1] + 0.03065999999999999, z_draw, base_p[3], base_p[4], base_p[5]), a=accel, v=vel)\n  movel(pose(base_p[0] + 0.16488, base_p[1] + 0.03065999999999999, z_draw, base_p[3], base_p[4], base_p[5]), a=accel, v=vel)\n  movel(pose(base_p[0] + 0.17664, base_p[1] + 0.028979999999999985, z_draw, base_p[3], base_p[4], base_p[5]), a=accel, v=vel)\n  movel(pose(base_p[0] + 0.1758, base_p[1] + 0.03653999999999999, z_draw, base_p[3], base_p[4], base_p[5]), a=accel, v=vel)\n  movel(pose(base_p[0] + 0.18336000000000002, base_p[1] + 0.04325999999999999, z_draw, base_p[3], base_p[4], base_p[5]), a=accel, v=vel)\n  movel(pose(base_p[0] + 0.19007999999999997, base_p[1] + 0.06005999999999999, z_draw, base_p[3], base_p[4], base_p[5]), a=accel, v=vel)\n  movel(pose(base_p[0] + 0.19007999999999997, base_p[1] + 0.08106, z_draw, base_p[3], base_p[4], base_p[5]), a=accel, v=vel)\n  movel(pose(base_p[0] + 0.18168, base_p[1] + 0.12894, z_draw, base_p[3], base_p[4], base_p[5]), a=accel, v=vel)\n  movel(pose(base_p[0] + 0.16656, base_p[1] + 0.15414, z_draw, base_p[3], base_p[4], base_p[5]), a=accel, v=vel)\n  movel(pose(base_p[0] + 0.16992000000000002, base_p[1] + 0.16254000000000002, z_draw, base_p[3], base_p[4], base_p[5]), a=accel, v=vel)\n  movel(pose(base_p[0] + 0.16739999999999997, base_p[1] + 0.17262, z_draw, base_p[3], base_p[4], base_p[5]), a=accel, v=vel)\n  movel(pose(base_p[0] + 0.16739999999999997, base_p[1] + 0.17262, z_move, base_p[3], base_p[4], base_p[5]), a=accel, v=vel)\n\n  # --- Path 19 ---\n  movel(pose(base_p[0] + 0.13632, base_p[1] + 0.17598000000000003, z_move, base_p[3], base_p[4], base_p[5]), a=accel, v=vel)\n  movel(pose(base_p[0] + 0.13632, base_p[1] + 0.17598000000000003, z_draw, base_p[3], base_p[4], base_p[5]), a=accel, v=vel)\n  movel(pose(base_p[0] + 0.13044, base_p[1] + 0.1743, z_draw, base_p[3], base_p[4], base_p[5]), a=accel, v=vel)\n  movel(pose(base_p[0] + 0.13044, base_p[1] + 0.15414, z_draw, base_p[3], base_p[4], base_p[5]), a=accel, v=vel)\n  movel(pose(base_p[0] + 0.11531999999999999, base_p[1] + 0.12642, z_draw, base_p[3], base_p[4], base_p[5]), a=accel, v=vel)\n  movel(pose(base_p[0] + 0.10523999999999999, base_p[1] + 0.07518, z_draw, base_p[3], base_p[4], base_p[5]), a=accel, v=vel)\n  movel(pose(base_p[0] + 0.10944, base_p[1] + 0.05081999999999999, z_draw, base_p[3], base_p[4], base_p[5]), a=accel, v=vel)\n  movel(pose(base_p[0] + 0.12204, base_p[1] + 0.03233999999999999, z_draw, base_p[3], base_p[4], base_p[5]), a=accel, v=vel)\n  movel(pose(base_p[0] + 0.10691999999999999, base_p[1] + 0.05081999999999999, z_draw, base_p[3], base_p[4], base_p[5]), a=accel, v=vel)\n  movel(pose(base_p[0] + 0.10188, base_p[1] + 0.08189999999999999, z_draw, base_p[3], base_p[4], base_p[5]), a=accel, v=vel)\n  movel(pose(base_p[0] + 0.10439999999999999, base_p[1] + 0.09617999999999999, z_draw, base_p[3], base_p[4], base_p[5]), a=accel, v=vel)\n  movel(pose(base_p[0] + 0.10272, base_p[1] + 0.06509999999999999, z_draw, base_p[3], base_p[4], base_p[5]), a=accel, v=vel)\n  movel(pose(base_p[0] + 0.12035999999999998, base_p[1] + 0.03233999999999999, z_draw, base_p[3], base_p[4], base_p[5]), a=accel, v=vel)\n  movel(pose(base_p[0] + 0.10944, base_p[1] + 0.022259999999999988, z_draw, base_p[3], base_p[4], base_p[5]), a=accel, v=vel)\n  movel(pose(base_p[0] + 0.13295999999999997, base_p[1] + 0.020579999999999987, z_draw, base_p[3], base_p[4], base_p[5]), a=accel, v=vel)\n  movel(pose(base_p[0] + 0.13716, base_p[1] + 0.026459999999999987, z_draw, base_p[3], base_p[4], base_p[5]), a=accel, v=vel)\n  movel(pose(base_p[0] + 0.13212000000000002, base_p[1] + 0.020579999999999987, z_draw, base_p[3], base_p[4], base_p[5]), a=accel, v=vel)\n  movel(pose(base_p[0] + 0.10944, base_p[1] + 0.02309999999999999, z_draw, base_p[3], base_p[4], base_p[5]), a=accel, v=vel)\n  movel(pose(base_p[0] + 0.12204, base_p[1] + 0.03233999999999999, z_draw, base_p[3], base_p[4], base_p[5]), a=accel, v=vel)\n  movel(pose(base_p[0] + 0.11783999999999999, base_p[1] + 0.023939999999999986, z_draw, base_p[3], base_p[4], base_p[5]), a=accel, v=vel)\n  movel(pose(base_p[0] + 0.13295999999999997, base_p[1] + 0.024779999999999986, z_draw, base_p[3], base_p[4], base_p[5]), a=accel, v=vel)\n  movel(pose(base_p[0] + 0.12035999999999998, base_p[1] + 0.027299999999999987, z_draw, base_p[3], base_p[4], base_p[5]), a=accel, v=vel)\n  movel(pose(base_p[0] + 0.12624, base_p[1] + 0.029819999999999985, z_draw, base_p[3], base_p[4], base_p[5]), a=accel, v=vel)\n  movel(pose(base_p[0] + 0.11028, base_p[1] + 0.06258, z_draw, base_p[3], base_p[4], base_p[5]), a=accel, v=vel)\n  movel(pose(base_p[0] + 0.11783999999999999, base_p[1] + 0.03989999999999999, z_draw, base_p[3], base_p[4], base_p[5]), a=accel, v=vel)\n  movel(pose(base_p[0] + 0.10691999999999999, base_p[1] + 0.059219999999999995, z_draw, base_p[3], base_p[4], base_p[5]), a=accel, v=vel)\n  movel(pose(base_p[0] + 0.11531999999999999, base_p[1] + 0.12642, z_draw, base_p[3], base_p[4], base_p[5]), a=accel, v=vel)\n  movel(pose(base_p[0] + 0.13044, base_p[1] + 0.15245999999999998, z_draw, base_p[3], base_p[4], base_p[5]), a=accel, v=vel)\n  movel(pose(base_p[0] + 0.12791999999999998, base_p[1] + 0.16674, z_draw, base_p[3], base_p[4], base_p[5]), a=accel, v=vel)\n  movel(pose(base_p[0] + 0.13295999999999997, base_p[1] + 0.17598000000000003, z_draw, base_p[3], base_p[4], base_p[5]), a=accel, v=vel)\n  movel(pose(base_p[0] + 0.14556, base_p[1] + 0.15918000000000002, z_draw, base_p[3], base_p[4], base_p[5]), a=accel, v=vel)\n  movel(pose(base_p[0] + 0.15732, base_p[1] + 0.16422000000000003, z_draw, base_p[3], base_p[4], base_p[5]), a=accel, v=vel)\n  movel(pose(base_p[0] + 0.14639999999999997, base_p[1] + 0.15918000000000002, z_draw, base_p[3], base_p[4], base_p[5]), a=accel, v=vel)\n  movel(pose(base_p[0] + 0.14639999999999997, base_p[1] + 0.15918000000000002, z_move, base_p[3], base_p[4], base_p[5]), a=accel, v=vel)\n\n  # --- Path 20 ---\n  movel(pose(base_p[0] + 0.14136, base_p[1] + 0.19025999999999998, z_move, base_p[3], base_p[4], base_p[5]), a=accel, v=vel)\n  movel(pose(base_p[0] + 0.14136, base_p[1] + 0.19025999999999998, z_draw, base_p[3], base_p[4], base_p[5]), a=accel, v=vel)\n  movel(pose(base_p[0] + 0.06323999999999999, base_p[1] + 0.06929999999999999, z_draw, base_p[3], base_p[4], base_p[5]), a=accel, v=vel)\n  movel(pose(base_p[0] + 0.10188, base_p[1] + 0.0945, z_draw, base_p[3], base_p[4], base_p[5]), a=accel, v=vel)\n  movel(pose(base_p[0] + 0.06743999999999999, base_p[1] + 0.06761999999999999, z_draw, base_p[3], base_p[4], base_p[5]), a=accel, v=vel)\n  movel(pose(base_p[0] + 0.06995999999999998, base_p[1] + 0.09029999999999999, z_draw, base_p[3], base_p[4], base_p[5]), a=accel, v=vel)\n  movel(pose(base_p[0] + 0.10607999999999998, base_p[1] + 0.12558, z_draw, base_p[3], base_p[4], base_p[5]), a=accel, v=vel)\n  movel(pose(base_p[0] + 0.13212000000000002, base_p[1] + 0.18354, z_draw, base_p[3], base_p[4], base_p[5]), a=accel, v=vel)\n  movel(pose(base_p[0] + 0.15647999999999998, base_p[1] + 0.19025999999999998, z_draw, base_p[3], base_p[4], base_p[5]), a=accel, v=vel)\n  movel(pose(base_p[0] + 0.19260000000000002, base_p[1] + 0.12306, z_draw, base_p[3], base_p[4], base_p[5]), a=accel, v=vel)\n  movel(pose(base_p[0] + 0.23376, base_p[1] + 0.07601999999999999, z_draw, base_p[3], base_p[4], base_p[5]), a=accel, v=vel)\n  movel(pose(base_p[0] + 0.22956000000000001, base_p[1] + 0.06761999999999999, z_draw, base_p[3], base_p[4], base_p[5]), a=accel, v=vel)\n  movel(pose(base_p[0] + 0.19260000000000002, base_p[1] + 0.09534, z_draw, base_p[3], base_p[4], base_p[5]), a=accel, v=vel)\n  movel(pose(base_p[0] + 0.19260000000000002, base_p[1] + 0.05837999999999999, z_draw, base_p[3], base_p[4], base_p[5]), a=accel, v=vel)\n  movel(pose(base_p[0] + 0.17748000000000003, base_p[1] + 0.033179999999999994, z_draw, base_p[3], base_p[4], base_p[5]), a=accel, v=vel)\n  movel(pose(base_p[0] + 0.18671999999999997, base_p[1] + 0.021419999999999988, z_draw, base_p[3], base_p[4], base_p[5]), a=accel, v=vel)\n  movel(pose(base_p[0] + 0.138, base_p[1] + 0.029819999999999985, z_draw, base_p[3], base_p[4], base_p[5]), a=accel, v=vel)\n  movel(pose(base_p[0] + 0.15983999999999998, base_p[1] + 0.03233999999999999, z_draw, base_p[3], base_p[4], base_p[5]), a=accel, v=vel)\n  movel(pose(base_p[0] + 0.16488, base_p[1] + 0.05165999999999999, z_draw, base_p[3], base_p[4], base_p[5]), a=accel, v=vel)\n  movel(pose(base_p[0] + 0.16319999999999998, base_p[1] + 0.025619999999999987, z_draw, base_p[3], base_p[4], base_p[5]), a=accel, v=vel)\n  movel(pose(base_p[0] + 0.17915999999999999, base_p[1] + 0.024779999999999986, z_draw, base_p[3], base_p[4], base_p[5]), a=accel, v=vel)\n  movel(pose(base_p[0] + 0.16319999999999998, base_p[1] + 0.027299999999999987, z_draw, base_p[3], base_p[4], base_p[5]), a=accel, v=vel)\n  movel(pose(base_p[0] + 0.16572, base_p[1] + 0.05249999999999999, z_draw, base_p[3], base_p[4], base_p[5]), a=accel, v=vel)\n  movel(pose(base_p[0] + 0.15647999999999998, base_p[1] + 0.031499999999999986, z_draw, base_p[3], base_p[4], base_p[5]), a=accel, v=vel)\n  movel(pose(base_p[0] + 0.138, base_p[1] + 0.031499999999999986, z_draw, base_p[3], base_p[4], base_p[5]), a=accel, v=vel)\n  movel(pose(base_p[0] + 0.13295999999999997, base_p[1] + 0.04661999999999999, z_draw, base_p[3], base_p[4], base_p[5]), a=accel, v=vel)\n  movel(pose(base_p[0] + 0.1338, base_p[1] + 0.026459999999999987, z_draw, base_p[3], base_p[4], base_p[5]), a=accel, v=vel)\n  movel(pose(base_p[0] + 0.1338, base_p[1] + 0.04577999999999999, z_draw, base_p[3], base_p[4], base_p[5]), a=accel, v=vel)\n  movel(pose(base_p[0] + 0.14051999999999998, base_p[1] + 0.027299999999999987, z_draw, base_p[3], base_p[4], base_p[5]), a=accel, v=vel)\n  movel(pose(base_p[0] + 0.18756, base_p[1] + 0.021419999999999988, z_draw, base_p[3], base_p[4], base_p[5]), a=accel, v=vel)\n  movel(pose(base_p[0] + 0.17748000000000003, base_p[1] + 0.03233999999999999, z_draw, base_p[3], base_p[4], base_p[5]), a=accel, v=vel)\n  movel(pose(base_p[0] + 0.19260000000000002, base_p[1] + 0.05837999999999999, z_draw, base_p[3], base_p[4], base_p[5]), a=accel, v=vel)\n  movel(pose(base_p[0] + 0.19260000000000002, base_p[1] + 0.0945, z_draw, base_p[3], base_p[4], base_p[5]), a=accel, v=vel)\n  movel(pose(base_p[0] + 0.22704000000000002, base_p[1] + 0.06846, z_draw, base_p[3], base_p[4], base_p[5]), a=accel, v=vel)\n  movel(pose(base_p[0] + 0.23292000000000002, base_p[1] + 0.07937999999999999, z_draw, base_p[3], base_p[4], base_p[5]), a=accel, v=vel)\n  movel(pose(base_p[0] + 0.18924000000000002, base_p[1] + 0.12894, z_draw, base_p[3], base_p[4], base_p[5]), a=accel, v=vel)\n  movel(pose(base_p[0] + 0.16656, base_p[1] + 0.18354, z_draw, base_p[3], base_p[4], base_p[5]), a=accel, v=vel)\n  movel(pose(base_p[0] + 0.16656, base_p[1] + 0.18354, z_move, base_p[3], base_p[4], base_p[5]), a=accel, v=vel)\n
  # --- End of Drawing ---
  # Lift the pen after the last path
  final_pose = get_actual_tcp_pose()
  movel(pose(final_pose[0], final_pose[1], z_move, final_pose[3], final_pose[4], final_pose[5]), a=accel, v=vel)
  textmsg("Drawing complete!")
  popup("Drawing complete!", "Info")
end
